// TwinCAT 3 PLC project Plc1
// ProgramVersion: 3.1.4022.2
// libraries:
//   log4TC, * (mbc engineering GmbH)
//   Tc2_Standard, * (Beckhoff Automation GmbH)
//   Tc2_System, * (Beckhoff Automation GmbH)
//   Tc3_Module, * (Beckhoff Automation GmbH)
// project tree:
//   / FB_LogTaskCycleTime.TcPOU, MAIN.TcPOU, PlcTask.TcTTO (not stored), PRG_SimulateLoad.TcPOU (not stored), PRG_SimulateLogs.TcPOU (not stored)

// ---- FB_LogTaskCycleTime.TcPOU
FUNCTION_BLOCK FB_LogTaskCycleTime
VAR_INPUT
	nCycleInterval	: UDINT;
END_VAR
VAR
	nTaskIndex		: DINT;
	nCycleCount		: UDINT;
	nExecTimeSum	: UDINT;
	nMaxExecTime	: UDINT := 0;
	nMinExecTime	: UDINT := 16#FFFFFFFF;
END_VAR
VAR_TEMP
	fExecAvg		: REAL;
END_VAR

nTaskIndex := Tc2_System.GETCURTASKINDEXEX();


nExecTimeSum := nExecTimeSum + _TaskInfo[nTaskIndex].LastExecTime;
nMaxExecTime := MAX(nMaxExecTime, _TaskInfo[nTaskIndex].LastExecTime);
nMinExecTime := MIN(nMinExecTime, _TaskInfo[nTaskIndex].LastExecTime);

nCycleCount := nCycleCount + 1;
IF nCycleCount > nCycleInterval THEN
	fExecAvg := UDINT_TO_REAL(nExecTimeSum) / UDINT_TO_REAL(nCycleCount);
	F_LogLA3(
		E_LogLevel.eDebug, 
		'FB_LogTaskCycleTime',
		'Cycle time statistic avg={avg}, min={min}, max={max}.',
		fExecAvg,
		nMinExecTime,
		nMaxExecTime
	);

	nCycleCount := 0;
	nMaxExecTime := 0;
	nMinExecTime := 16#FFFFFFFF;
	nExecTimeSum := 0;
END_IF

END_FUNCTION_BLOCK

// ---- MAIN.TcPOU
PROGRAM MAIN
VAR
	fbCycleTimeLogger	: FB_LogTaskCycleTime := (nCycleInterval:=1000);
END_VAR

IF _TaskInfo[1].FirstCycle THEN
	// Change AMS id if log service runs on different server than
	// plc. Remove if plc and service runs on the same machine.
	PRG_TaskLog.Init('192.168.56.1.1.1');
	F_Log(E_LogLevel.eInfo, 'Plc started.');
END_IF

// simulates load on the task
PRG_SimulateLoad();

// simulate logs
PRG_SimulateLogs();

// logs the cycle time statistics
fbCycleTimeLogger();

PRG_TaskLog.Call();

END_PROGRAM
